{attribute 'linkalways'} 
{attribute 'no_explicit_call' := 'This FB is a CLASS and must be accessed using methods or properties'}
{attribute 'enable_dynamic_creation'}
FUNCTION_BLOCK Node_RGBA_BLACK EXTENDS VisionNode
VAR
    out : _TcVnVector4_LREAL;
END_VAR

METHOD PUBLIC  Clone : I_Node
VAR
	pNode : POINTER TO Node_RGBA_BLACK;
END_VAR
pNode := __NEW(Node_RGBA_BLACK);
Clone := pNode^;
END_METHOD

METHOD FB_init : BOOL
VAR_INPUT
	bInitRetains : BOOL; // if TRUE, the retain variables are initialized (warm start / cold start)
	bInCopyCode : BOOL;  // if TRUE, the instance afterwards gets moved into the copy code (online change)
END_VAR
AddOutput('out', out);
END_METHOD

METHOD PROTECTED OnExecute
out.Value := GVL_COLOURS.RGBA_BLACK;
END_METHOD

METHOD PUBLIC PreExecutionCheck
VAR_INPUT
	Check : I_PreExecutionChecks;
END_VAR
END_METHOD

END_FUNCTION_BLOCK

(* stored: Version 1.1.0.1, ProductVersion 3.1.4024.13
   POU Node_RGBA_BLACK: Id {7c4d575f-92cc-0fa8-2a59-c6ca3933c566}, SpecialFunc None
   Folder Constructor: Id {b26a70ad-af83-0b84-1358-69b607bb5f8b}
   Method Clone: Id {ed4fd8f4-5e11-0e8f-25bf-2e56a18e1295}
   Method FB_init: Id {0a61193d-d84a-0e1e-1dcc-b20fd661be90}
   Method OnExecute: Id {21d19c37-6014-0322-321c-5dc117a8edeb}
   Method PreExecutionCheck: Id {8de6fd09-1df7-0a54-0aef-c95cf036499b} *)
